{attribute addProperty BoxType "EL2252--0000"}
{attribute addProperty Id "DC_Sync_ActivateAT %Q*DC_Sync_Activate_03B9C976810DC_Sync_StartAT %Q*DC_Sync_Start_771C156B3240ChannelAT %Q*ARRAY[0..1] OF Channel_7F374EB01620WcStateAT %I*WcState_28A8677510.1250InfoDataAT %I*InfoData_7231B2DD80100"}
{attribute addProperty CRC "197302945"}
{attribute addProperty SizeInBites "137"}
{attribute addProperty SizeInBytes "17.125"}
TYPE EL2252_3BE0B4B7 :
STRUCT
	{attribute addProperty Name "DC_Sync_Activate"}
	DC_Sync_Activate : DC_Sync_Activate_03B9C976;
	{attribute addProperty Name "DC_Sync_Start"}
	DC_Sync_Start : DC_Sync_Start_771C156B;
	{attribute addProperty Name "Channel"}
	Channel : ARRAY[0..1] OF Channel_7F374EB0;
	{attribute addProperty Name "WcState"}
	WcState : WcState_28A86775;
	{attribute addProperty Name "InfoData"}
	InfoData : InfoData_7231B2DD;
END_STRUCT
END_TYPE

(* stored: Version 1.2.0.0, ProductVersion 3.1.4024.9
   DUT EL2252_3BE0B4B7: Id {fd9ed173-09cc-437d-8de9-ded060c23a8c} *)
